// TIA Portal V17 export
// export: Created 2025-03-05T08:02:29.2624853Z, ExportSetting WithDefaults, DisplayName Totally Integrated Automation Portal, DisplayVersion V17 Update 8, DisplayName TIA Portal Openness, DisplayVersion V17 Update 8, DisplayName TIA Portal Version Control Interface, DisplayVersion V17, DisplayName SINAMICS Startdrive Advanced, DisplayVersion V17 SP2, DisplayName SINAMICS Startdrive G110M, G120, G120C, G120D, G120P, G115D, DisplayVersion V17 SP2, DisplayName SINAMICS Startdrive G130, G150, S120, S150, SINAMICS MV, S210, DisplayVersion V17 SP2, DisplayName STEP 7 Professional, DisplayVersion V17 Update 8, DisplayName SINUMERIK ONE STEP 7 Toolbox, DisplayVersion V17 Update 12, DisplayName SINUMERIK 840D sl STEP 7 Toolbox, DisplayVersion V17 Update 12, DisplayName STEP 7 Safety, DisplayVersion V17 Update 6, DisplayName WinCC Advanced, DisplayVersion V17 Update 8
TYPE "POWDER FEEDER INTERLOCK INPUT"
// stored: IsFailsafeCompliant false
   STRUCT
      i_uiOperationMode_Line1 : Word;   // Current Line Operation Mode 0 = Stand Alone, 1 = On Off Remote 2 = UDP, 3 = Profibus, 5 = Device Net / current line operation mode 0 = Standalone, 1 = OnOffRemote 2 = UDP, 3 = Profibus, 4 = ProfiNet, 5 = DeviceNet
      i_uiOperationMode_Line2 : Word;   // Current Line Operation Mode 0 = Stand Alone, 1 = On Off Remote 2 = UDP, 3 = Profibus, 5 = Device Net / current line operation mode 0 = Standalone, 1 = OnOffRemote 2 = UDP, 3 = Profibus, 4 = ProfiNet, 5 = DeviceNet
      i_uiFeederState_Line1 : Word;   // Current Feeder Line StateCG_Feedfun_Disabled=0, Cg_Ready_Start=1,Cg_Wait_To_Eestablish=2, Feedfunc_Ready_Start=3,Feedfun_Running=4, Feedfun_Wait_To_Zero=5 / current feeder line state CG_FEEDFUN_DISABLED=0, CG_READY_START=1, CG_WAIT_TO_ESTABLISH=2, FEEDFUNC_READY_START=3, FEEDFUN_RUNNING=4, FEEDFUN_WAIT_TO_ZERO=5
      i_uiFeederState_Line2 : Word;   // Current Feeder Line StateCG_Feedfun_Disabled=0, Cg_Ready_Start=1,Cg_Wait_To_Establish=2, Feedfunc_Ready_Start=3,Feedfun_Running=4, Feedfun_Wait_To_Zero=5 / current feeder line state CG_FEEDFUN_DISABLED=0, CG_READY_START=1, CG_WAIT_TO_ESTABLISH=2, FEEDFUNC_READY_START=3, FEEDFUN_RUNNING=4, FEEDFUN_WAIT_TO_ZERO=5
      i_fOperationModeMatched_Line1 : Bool;   // O_UiOperationMode Is Equal To Feeder Line Operation Mode / o_uiOperationMode is equal to feeder line operation mode
      i_fOperationModeMatched_Line2 : Bool;   // O_UiOperationMode Is Equal To Feeder Line Operation Mode / o_uiOperationMode is equal to feeder line operation mode
      i_fFeedingMode_Line1 : Bool;   // 0 = Volumetric (For Twin 150 Always Volumetric) 1 = Gravimetric / 0 = volumetric (for Twin 150 always volumetric), 1 = gravimetric
      i_fFeedingMode_Line2 : Bool;   // 0 = Volumetric (For Twin 150 Always Volumetric) 1 = Gravimetric / 0 = volumetric (for Twin 150 always volumetric), 1 = gravimetric
      i_fFeederReady_Line1 : Bool;   // No Shutdown Present / No shutdown present
      i_fFeederReady_Line2 : Bool;   // No Shutdown Present / No shutdown present
      i_fTareDone_Line1 : Bool;   // N/a For Twin 150 / n/a for Twin 150
      i_fTareDone_Line2 : Bool;   // N/a For Twin 150 / n/a for Twin 150
      i_fCalibDone_Line1 : Bool;   // N/a For Twin 150 / n/a for Twin 150
      i_fCalibDone_Line2 : Bool;   // N/a For Twin 150 / n/a for Twin 150
      i_fCarrierGasSelected_Line1 : Bool;   // 0 = Argon Selected, 1 = Nitrogen Selected / 0 = Argon selected, 1 = Nitrogen selected
      i_fCarrierGasSelected_Line2 : Bool;   // 0 = Argon Selected, 1 = Nitrogen Selected / 0 = Argon selected, 1 = Nitrogen selected
      i_fUnitSelected_Line1 : Bool;   // 0 = Metric Units, 1 = SI / 0 = metric units, 1 = SI
      i_fUnitSelected_Line2 : Bool;   // 0 = Metric Units, 1 = SI / 0 = metric units, 1 = SI
      i_fPowderLineClogged_Line1 : Bool;   // 0 = Line Not Clogged, 1 = Line Is Clogged (Overpressure) / 0 = line not clogged, 1 = line is clogged (overpressure)
      i_fPowderLineClogged_Line2 : Bool;   // 0 = Line Not Clogged, 1 = Line Is Clogged (Overpressure) / 0 = line not clogged, 1 = line is clogged (overpressure)
      i_fShutdownFromPf_Line1 : Bool;   // 0 = No Shutdown Present, 1 = Shutdown Present For Feeder Line / 0 = no shutdown present, 1 = shutdown present for feeder line
      i_fShutdownFromPf_Line2 : Bool;   // 0 = No Shutdown Present, 1 = Shutdown Present For Feeder Line / 0 = no shutdown present, 1 = shutdown present for feeder line
      i_fWarningFromPF_Line1 : Bool;   // 0 = No Warning Present, 1 = Warning Present For Feeder Line / 0 = no warning present, 1 = warning present for feeder line
      i_fWarningFromPF_Line2 : Bool;   // 0 = No Warning Present, 1 = Warning Present For Feeder Line / 0 = no warning present, 1 = warning present for feeder line
      i_fDiskStatus_Line1 : Bool;   // 0 = Disk Motor Not Ready, 1 = Disk Motor Plugged In And Ready / 0 = disk motor not ready, 1 = disk motor plugged in and ready
      i_fDiskStatus_Line2 : Bool;   // 0 = Disk Motor Not Ready, 1 = Disk Motor Plugged In And Ready / 0 = disk motor not ready, 1 = disk motor plugged in and ready
      i_fStirrerStatus_Line1 : Bool;   // 0 = Stirrer Motor Not Ready, 1 = Stirrer Is Plugged In And Ready / 0 = stirrer motor not ready, 1 = stirrer is plugged in and ready
      i_fStirrerStatus_Line2 : Bool;   // 0 = Stirrer Motor Not Ready, 1 = Stirrer Is Plugged In And Ready / 0 = stirrer motor not ready, 1 = stirrer is plugged in and ready
      i_fCarriergasStatus_Line1 : Bool;   // 0 = Carrier Gas Is Off, 1 = Carrier Gas Is Running / 0 = carriergas is off, 1 = carriergas is running
      i_fCarriergasStatus_Line2 : Bool;   // 0 = Carrier Gas Is Off, 1 = Carrier Gas Is Running / 0 = carriergas is off, 1 = carriergas is running
      i_fCommunicationOK_Line1 : Bool;   // 1 = Communication Running / 1 = Communication running
      i_fCommunicationOK_Line2 : Bool;   // 1 = Communication Running / 1 = Communication running
      i_fCarriergasLeLL_Line1 : Bool;   // 0 = Carrier Gas Flow > LL Limit, 1 = Carrier Gas Flow < LL Limit / 0 = carriergas flow > LL limit, 1 = carriergas flow < LL limit
      i_fCarriergasLeLL_Line2 : Bool;   // 0 = Carrier Gas Flow > LL Limit, 1 = Carrier Gas Flow < LL Limit / 0 = carriergas flow > LL limit, 1 = carriergas flow < LL limit
      i_fDiskSpeedLeLL_Line1 : Bool;   // 0 = Disk Speed > LL Limit, 1 = Disk Speed < LL Limit / 0 = disk speed > LL limit, 1 = disk speed < LL limit
      i_fDiskSpeedLeLL_Line2 : Bool;   // 0 = Disk Speed > LL Limit, 1 = Disk Speed < LL Limit / 0 = disk speed > LL limit, 1 = disk speed < LL limit
      i_fStirrerSpeedLeLL_Line1 : Bool;   // 0 = Stirrer Speed > LL Limit, 1 = Stirrer Speed < LL Limit / 0 = stirrer speed > LL limit, 1 = stirrer speed < LL limit
      i_fStirrerSpeedLeLL_Line2 : Bool;   // 0 = Stirrer Speed > LL Limit, 1 = Stirrer Speed < LL Limit / 0 = stirrer speed > LL limit, 1 = stirrer speed < LL limit
      i_fFeedrateLeLL_Line1 : Bool;   // N/a For Twin 150 / n/a for Twin 150
      i_fFeedrateLeLL_Line2 : Bool;   // N/a For Twin 150 / n/a for Twin 150
      i_fPowderLevelLeLL_Line1 : Bool;   // N/a For Twin 150 / n/a for Twin 150
      i_fPowderLevelLeLL_Line2 : Bool;   // N/a For Twin 150 / n/a for Twin 150
      i_fCarriergasLeL_Line1 : Bool;   // 0 = Carrier Gas Flow > L Limit, 1 = Carrier Gas Flow < L Limit / 0 = carriergas flow > L limit, 1 = carriergas flow < L limit
      i_fCarriergasLeL_Line2 : Bool;   // 0 = Carrier Gas Flow > L Limit, 1 = Carrier Gas Flow < L Limit / 0 = carriergas flow > L limit, 1 = carriergas flow < L limit
      i_fDiskSpeedLeL_Line1 : Bool;   // 0 = Disk Speed > L Limit, 1 = Disk Speed < L Limit / 0 = disk speed > L limit, 1 = disk speed < L limit
      i_fDiskSpeedLeL_Line2 : Bool;   // 0 = Disk Speed > L Limit, 1 = Disk Speed < L Limit / 0 = disk speed > L limit, 1 = disk speed < L limit
      i_fStirrerSpeedLeL_Line1 : Bool;   // 0 = Stirrer Speed > L Limit, 1 = Stirrer Speed < L Limit / 0 = Stirrer speed > L limit, 1 = Stirrer speed < L limit
      i_fStirrerSpeedLeL_Line2 : Bool;   // 0 = Stirrer Speed > L Limit, 1 = Stirrer Speed < L Limit / 0 = Stirrer speed > L limit, 1 = Stirrer speed < L limit
      i_fFeedrateLeL_Line1 : Bool;   // N/a For Twin 150 / n/a for Twin 150
      i_fFeedrateLeL_Line2 : Bool;   // N/a For Twin 150 / n/a for Twin 150
      i_fPowderLevelLeL_Line1 : Bool;   // N/a For Twin 150 / n/a for Twin 150
      i_fPowderLevelLeL_Line2 : Bool;   // N/a For Twin 150 / n/a for Twin 150
      i_fCarriergasGrH_Line1 : Bool;   // 0 = Carrier Gas Flow < H Limit, 1 = Carrier Gas Flow > H Limit / 0 = carriergas flow < H limit, 1 = carriergas flow > H limit
      i_fCarriergasGrH_Line2 : Bool;   // 0 = Carrier Gas Flow < H Limit, 1 = Carrier Gas Flow > H Limit / 0 = carriergas flow < H limit, 1 = carriergas flow > H limit
      i_fDiskSpeedGrH_Line1 : Bool;   // 0 = Disk Speed < H Limit, 1 = Disk Speed > H Limit / 0 = disk speed < H limit, 1 = disk speed > H limit
      i_fDiskSpeedGrH_Line2 : Bool;   // 0 = Disk Speed < H Limit, 1 = Disk Speed > H Limit / 0 = disk speed < H limit, 1 = disk speed > H limit
      i_fStirrerSpeedGrH_Line1 : Bool;   // 0 = Stirrer Speed < H Limit, 1 = Stirrer Speed > H Limit / 0 = Stirrer speed < H limit, 1 = Stirrer speed > H limit
      i_fStirrerSpeedGrH_Line2 : Bool;   // 0 = Stirrer Speed < H Limit, 1 = Stirrer Speed > H Limit / 0 = Stirrer speed < H limit, 1 = Stirrer speed > H limit
      i_fFeedrateGrH_Line1 : Bool;   // N/a For Twin 150 / n/a for Twin 150
      i_fFeedrateGrH_Line2 : Bool;   // N/a For Twin 150 / n/a for Twin 150
      i_fCarriergasGrHH_Line1 : Bool;   // 0 = Carrier Gas Flow < HH Limit, 1 = Carriergas Flow > HH Limit / 0 = carriergas flow < HH limit, 1 = carriergas flow > HH limit
      i_fCarriergasGrHH_Line2 : Bool;   // 0 = Carrier Gas Flow < HH Limit, 1 = Carriergas Flow > HH Limit / 0 = carriergas flow < HH limit, 1 = carriergas flow > HH limit
      i_fDiskSpeedGrHH_Line1 : Bool;   // 0 = Disk Speed < HH Limit, 1 = Disk Speed > HH Limit / 0 = disk speed < HH limit, 1 = disk speed > HH limit
      i_fDiskSpeedGrHH_Line2 : Bool;   // 0 = Disk Speed < HH Limit, 1 = Disk Speed > HH Limit / 0 = disk speed < HH limit, 1 = disk speed > HH limit
      i_fStirrerSpeedGrHH_Line1 : Bool;   // 0 = Stirrer Speed < HH Limit, 1 = Stirrer Speed > HH Limit / 0 = Stirrer speed < HH limit, 1 = Stirrer speed > HH limit
      i_fStirrerSpeedGrHH_Line2 : Bool;   // 0 = Stirrer Speed < HH Limit, 1 = Stirrer Speed > HH Limit / 0 = Stirrer speed < HH limit, 1 = Stirrer speed > HH limit
      i_fHopperTempGrHH_Line1 : Bool;   // 0 = Hopper Temperature < HH Limit 110ºC, 1 = Hopper Temperature > HH Limit 110ºC / 0 = Hopper temperature < 110 °C, 1 = Hopper temperature > 110 °C
      i_fHopperTempGrHH_Line2 : Bool;   // 0 = Hopper Temperature < HH Limit 110ºC, 1 = Hopper Temperature > HH Limit 110ºC / 0 = Hopper temperature < 110 °C, 1 = Hopper temperature > 110 °C
      i_fFeedrateGrHH_Line1 : Bool;   // N/a For Twin 150 / 0 = Feedrate < HH limit, 1 = Feedrate > HH limit
      i_fFeedrateGrHH_Line2 : Bool;   // N/a For Twin 150 / 0 = Feedrate < HH limit, 1 = Feedrate > HH limit
      i_fCarriergasInletPressureTooLow_Line1 : Bool;   // 0 = Carrier Gas Pressure OK. 1 = Carriergas Pressure Too Low (Only If Pressure Switch Available) / 0 = carriergas pressure OK, 1 = carriergas pressure too low (only if pressure switch available)
      i_fCarriergasInletPressureTooLow_Line2 : Bool;   // 0 = Carrier Gas Pressure OK. 1 = Carriergas Pressure Too Low (Only If Pressure Switch Available) / 0 = carriergas pressure OK, 1 = carriergas pressure too low (only if pressure switch available)
      Spare_0 : Bool;   // Spare
      Spare_1 : Bool;   // Spare
      Spare_2 : Bool;   // Spare
      Spare_3 : Bool;   // Spare
      i_f_OptionHeatingAvailable_Line1 : Bool;   // 1 = Option Available / 1 = option available
      i_f_OptionHeatingAvailable_Line2 : Bool;   // 1 = Option Available / 1 = option available
      Spare_4 : Bool;   // Spare
      Spare_5 : Bool;   // Spare
      Spare_6 : Bool;   // Spare
      Spare_7 : Bool;   // Spare
      Spare_8 : Bool;   // Spare
      Spare_9 : Bool;   // Spare
      Spare_Byte_1 : Byte;   // Spare
      Spare_Byte_2 : Byte;   // Spare
      "Actual PF Values" : Struct
         i_rCarriergasActual_Line1 : Real;   // Actual Value Carriergas Flow (NLPM) / actual value carriergas flow [NLPM]
         i_rCarriergasActual_Line2 : Real;   // Actual Value Carriergas Flow (NLPM) / actual value carriergas flow [NLPM]
         i_rDiskActual_Line1 : Real;   // Actual Value Disk Speed (%) / actual value disk speed [%]
         i_rDiskActual_Line2 : Real;   // Actual Value Disk Speed (%) / actual value disk speed [%]
         i_rStirrerActual_Line1 : Real;   // Actual Value Stirrer Speed (%) / actual value stirrer speed [%]
         i_rStirrerActual_Line2 : Real;   // Actual Value Stirrer Speed (%) / actual value stirrer speed [%]
         i_rFeedrateActual_Line1 : Real;   // N/A For Twin 150 / n/a for Twin 150
         i_rFeedrateActual_Line2 : Real;   // N/A For Twin 150 / n/a for Twin 150
         i_rHopperTempActual_Line1 : Real;   // Actual Value Hopper Temperature (ºC) / actual value hopper temperature [°C]
         i_rHopperTempActual_Line2 : Real;   // Actual Value Hopper Temperature (ºC) / actual value hopper temperature [°C]
         i_rHopperPressureActual_Line1 : Real;   // Actual Value Hopper Pressure (Bar) / actual value hopper pressure [Bar]
         i_rHopperPressureActual_Line2 : Real;   // Actual Value Hopper Pressure (Bar) / actual value hopper pressure [Bar]
         i_rWeightActual_Line1 : Real;   // N/A For Twin 150 / n/a for Twin 150
         i_rWeightActual_Line2 : Real;   // N/A For Twin 150 / n/a for Twin 150
         i_rPowderFactorActual_Line1 : Real;   // N/A For Twin 150 / n/a for Twin 150
         i_rPowderFactorActual_Line2 : Real;   // N/A For Twin 150 / n/a for Twin 150
      END_STRUCT;
   END_STRUCT;
END_TYPE
